// TIA Portal V17 export
// export: Created 2023-05-12T10:40:25.6107869Z, DisplayName Totally Integrated Automation Portal, DisplayVersion V17 Update 4, DisplayName TIA Portal Openness, DisplayVersion V17 Update 4, DisplayName TIA Portal Version Control Interface, DisplayVersion V17, DisplayName STEP 7 Professional, DisplayVersion V17 Update 4, DisplayName STEP 7 Safety, DisplayVersion V17, DisplayName WinCC Advanced / Unified PC, DisplayVersion V17 Update 4
FUNCTION_BLOCK "FB_EM_InputConditioning"   // FB19, LAD
{ S7_Optimized_Access := 'TRUE' }
VERSION : 0.1
// stored: AutoNumber true, CodeModifiedDate 2023-05-12T12:59:41.6492354Z, CompileDate 2023-05-12T12:59:41.6492354Z, CreationDate 2023-05-08T12:19:11.3376827Z, DownloadWithoutReinit false, HandleErrorsWithinBlock false, InterfaceModifiedDate 2023-05-12T12:59:19.7337351Z, IsConsistent true, IsIECCheckEnabled false, IsKnowHowProtected false, IsRetainMemResEnabled false, IsWriteProtected false, LibraryConformanceStatus Warning: The object contains access to global data blocks., MemoryReserve 100, ModifiedDate 2023-05-12T12:59:41.6492354Z, ParameterModified 2022-09-13T10:25:33.4387708Z, PLCSimAdvancedSupport true, SetENOAutomatically false, StructureModified 2023-05-12T12:59:19.7337351Z, UDAEnableTagReadback false
   VAR
      "TT01_TempZasil_K-22/4_Inst" { S7_SetPoint := 'True'} : "FB_CM_MeasurementPoint";
      "TT02_TempPowr_K-22/4_Inst" { S7_SetPoint := 'True'} : "FB_CM_MeasurementPoint";
      TT04_TempPowr_Os_Rzepichy_Inst { S7_SetPoint := 'True'} : "FB_CM_MeasurementPoint";
      TT06_TempPowr_Zabianka_Inst { S7_SetPoint := 'True'} : "FB_CM_MeasurementPoint";
      "PT01_CisnZasil_ K-22/4_Inst" { S7_SetPoint := 'True'} : "FB_CM_MeasurementPoint";
      "PT02_CisnPowr_ K-22/4_Inst" { S7_SetPoint := 'True'} : "FB_CM_MeasurementPoint";
      PT03_CisnZasil_Os_Rzepichy_Inst { S7_SetPoint := 'True'} : "FB_CM_MeasurementPoint";
      PT04_CisnPowr_Os_Rzepichy_Inst { S7_SetPoint := 'True'} : "FB_CM_MeasurementPoint";
      PT05_CisnZasil_Zabianka_Inst { S7_SetPoint := 'True'} : "FB_CM_MeasurementPoint";
      PT06_CisnPowr_Zabianka_Inst { S7_SetPoint := 'True'} : "FB_CM_MeasurementPoint";
      TTs_TempSzafy_Inst { S7_SetPoint := 'True'} : "FB_CM_MeasurementPoint";
      TTk_TempKom_Inst { S7_SetPoint := 'True'} : "FB_CM_MeasurementPoint";
      TTz_TempZewn_Inst { S7_SetPoint := 'True'} : "FB_CM_MeasurementPoint";
      FT01_Przeplyw_Inst { S7_SetPoint := 'True'} : "FB_CM_MeasurementPoint";
      Rezerwa1_Inst { S7_SetPoint := 'True'} : "FB_CM_MeasurementPoint";
      Rezerwa2_Inst { S7_SetPoint := 'True'} : "FB_CM_MeasurementPoint";
   END_VAR
BEGIN

REGION Network 1: TT01_TempZasil_K-22/4 - Temperatura zasilania z K-22/4
   // TT01_TempZasil_K-22/4 - Temperatura zasilania z K-22/4
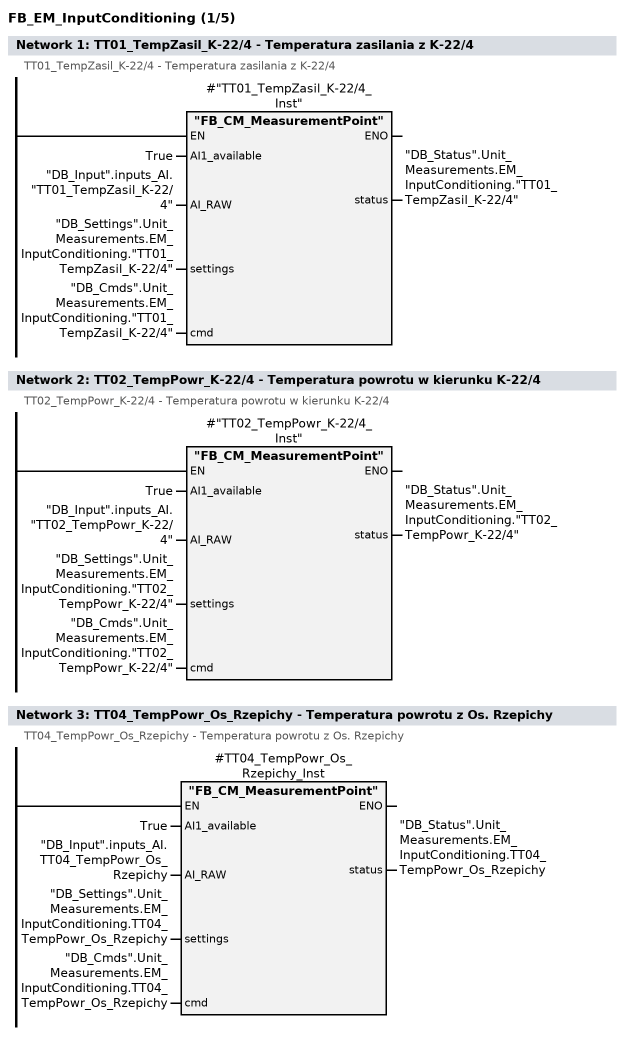
   RUNG wire#powerrail
      #"TT01_TempZasil_K-22/4_Inst"(AI1_available := True, AI_RAW := "DB_Input".inputs_AI."TT01_TempZasil_K-22/4", settings := "DB_Settings".Unit_Measurements.EM_InputConditioning."TT01_TempZasil_K-22/4", cmd := "DB_Cmds".Unit_Measurements.EM_InputConditioning."TT01_TempZasil_K-22/4", status => "DB_Status".Unit_Measurements.EM_InputConditioning."TT01_TempZasil_K-22/4")
   END_RUNG
   // the same network as SCL:
   #"TT01_TempZasil_K-22/4_Inst"(AI1_available := True,   // "FB_CM_MeasurementPoint"
                           AI_RAW := "DB_Input".inputs_AI."TT01_TempZasil_K-22/4",
                           settings := "DB_Settings".Unit_Measurements.EM_InputConditioning."TT01_TempZasil_K-22/4",
                           cmd := "DB_Cmds".Unit_Measurements.EM_InputConditioning."TT01_TempZasil_K-22/4",
                           status => "DB_Status".Unit_Measurements.EM_InputConditioning."TT01_TempZasil_K-22/4");
END_REGION

REGION Network 2: TT02_TempPowr_K-22/4 - Temperatura powrotu w kierunku K-22/4
   // TT02_TempPowr_K-22/4 - Temperatura powrotu w kierunku K-22/4
   RUNG wire#powerrail
      #"TT02_TempPowr_K-22/4_Inst"(AI1_available := True, AI_RAW := "DB_Input".inputs_AI."TT02_TempPowr_K-22/4", settings := "DB_Settings".Unit_Measurements.EM_InputConditioning."TT02_TempPowr_K-22/4", cmd := "DB_Cmds".Unit_Measurements.EM_InputConditioning."TT02_TempPowr_K-22/4", status => "DB_Status".Unit_Measurements.EM_InputConditioning."TT02_TempPowr_K-22/4")
   END_RUNG
   // the same network as SCL:
   #"TT02_TempPowr_K-22/4_Inst"(AI1_available := True,   // "FB_CM_MeasurementPoint"
                           AI_RAW := "DB_Input".inputs_AI."TT02_TempPowr_K-22/4",
                           settings := "DB_Settings".Unit_Measurements.EM_InputConditioning."TT02_TempPowr_K-22/4",
                           cmd := "DB_Cmds".Unit_Measurements.EM_InputConditioning."TT02_TempPowr_K-22/4",
                           status => "DB_Status".Unit_Measurements.EM_InputConditioning."TT02_TempPowr_K-22/4");
END_REGION

REGION Network 3: TT04_TempPowr_Os_Rzepichy - Temperatura powrotu z Os. Rzepichy
   // TT04_TempPowr_Os_Rzepichy - Temperatura powrotu z Os. Rzepichy
   RUNG wire#powerrail
      #TT04_TempPowr_Os_Rzepichy_Inst(AI1_available := True, AI_RAW := "DB_Input".inputs_AI.TT04_TempPowr_Os_Rzepichy, settings := "DB_Settings".Unit_Measurements.EM_InputConditioning.TT04_TempPowr_Os_Rzepichy, cmd := "DB_Cmds".Unit_Measurements.EM_InputConditioning.TT04_TempPowr_Os_Rzepichy, status => "DB_Status".Unit_Measurements.EM_InputConditioning.TT04_TempPowr_Os_Rzepichy)
   END_RUNG
   // the same network as SCL:
   #TT04_TempPowr_Os_Rzepichy_Inst(AI1_available := True,   // "FB_CM_MeasurementPoint"
                           AI_RAW := "DB_Input".inputs_AI.TT04_TempPowr_Os_Rzepichy,
                           settings := "DB_Settings".Unit_Measurements.EM_InputConditioning.TT04_TempPowr_Os_Rzepichy,
                           cmd := "DB_Cmds".Unit_Measurements.EM_InputConditioning.TT04_TempPowr_Os_Rzepichy,
                           status => "DB_Status".Unit_Measurements.EM_InputConditioning.TT04_TempPowr_Os_Rzepichy);
END_REGION

REGION Network 4: TT06_TempPowr_Zabianka - Temperatura powrotu z Żabianka
   // TT06_TempPowr_Zabianka - Temperatura powrotu z Żabianka
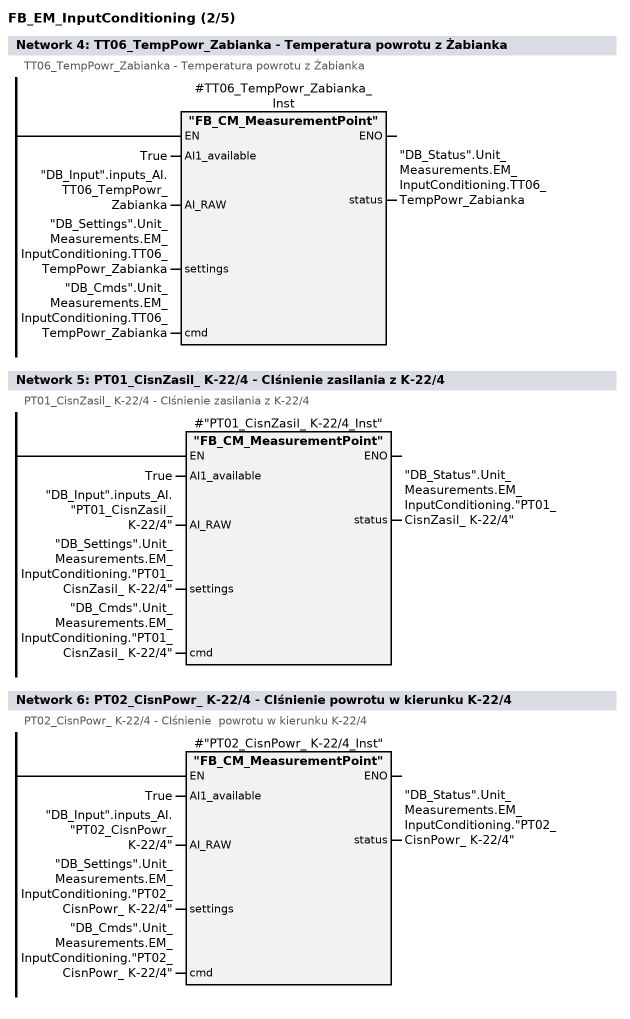
   RUNG wire#powerrail
      #TT06_TempPowr_Zabianka_Inst(AI1_available := True, AI_RAW := "DB_Input".inputs_AI.TT06_TempPowr_Zabianka, settings := "DB_Settings".Unit_Measurements.EM_InputConditioning.TT06_TempPowr_Zabianka, cmd := "DB_Cmds".Unit_Measurements.EM_InputConditioning.TT06_TempPowr_Zabianka, status => "DB_Status".Unit_Measurements.EM_InputConditioning.TT06_TempPowr_Zabianka)
   END_RUNG
   // the same network as SCL:
   #TT06_TempPowr_Zabianka_Inst(AI1_available := True,   // "FB_CM_MeasurementPoint"
                           AI_RAW := "DB_Input".inputs_AI.TT06_TempPowr_Zabianka,
                           settings := "DB_Settings".Unit_Measurements.EM_InputConditioning.TT06_TempPowr_Zabianka,
                           cmd := "DB_Cmds".Unit_Measurements.EM_InputConditioning.TT06_TempPowr_Zabianka,
                           status => "DB_Status".Unit_Measurements.EM_InputConditioning.TT06_TempPowr_Zabianka);
END_REGION

REGION Network 5: PT01_CisnZasil_ K-22/4 - CIśnienie zasilania z K-22/4
   // PT01_CisnZasil_ K-22/4 - CIśnienie zasilania z K-22/4
   RUNG wire#powerrail
      #"PT01_CisnZasil_ K-22/4_Inst"(AI1_available := True, AI_RAW := "DB_Input".inputs_AI."PT01_CisnZasil_ K-22/4", settings := "DB_Settings".Unit_Measurements.EM_InputConditioning."PT01_CisnZasil_ K-22/4", cmd := "DB_Cmds".Unit_Measurements.EM_InputConditioning."PT01_CisnZasil_ K-22/4", status => "DB_Status".Unit_Measurements.EM_InputConditioning."PT01_CisnZasil_ K-22/4")
   END_RUNG
   // the same network as SCL:
   #"PT01_CisnZasil_ K-22/4_Inst"(AI1_available := True,   // "FB_CM_MeasurementPoint"
                           AI_RAW := "DB_Input".inputs_AI."PT01_CisnZasil_ K-22/4",
                           settings := "DB_Settings".Unit_Measurements.EM_InputConditioning."PT01_CisnZasil_ K-22/4",
                           cmd := "DB_Cmds".Unit_Measurements.EM_InputConditioning."PT01_CisnZasil_ K-22/4",
                           status => "DB_Status".Unit_Measurements.EM_InputConditioning."PT01_CisnZasil_ K-22/4");
END_REGION

REGION Network 6: PT02_CisnPowr_ K-22/4 - CIśnienie powrotu w kierunku K-22/4
   // PT02_CisnPowr_ K-22/4 - CIśnienie  powrotu w kierunku K-22/4
   RUNG wire#powerrail
      #"PT02_CisnPowr_ K-22/4_Inst"(AI1_available := True, AI_RAW := "DB_Input".inputs_AI."PT02_CisnPowr_ K-22/4", settings := "DB_Settings".Unit_Measurements.EM_InputConditioning."PT02_CisnPowr_ K-22/4", cmd := "DB_Cmds".Unit_Measurements.EM_InputConditioning."PT02_CisnPowr_ K-22/4", status => "DB_Status".Unit_Measurements.EM_InputConditioning."PT02_CisnPowr_ K-22/4")
   END_RUNG
   // the same network as SCL:
   #"PT02_CisnPowr_ K-22/4_Inst"(AI1_available := True,   // "FB_CM_MeasurementPoint"
                           AI_RAW := "DB_Input".inputs_AI."PT02_CisnPowr_ K-22/4",
                           settings := "DB_Settings".Unit_Measurements.EM_InputConditioning."PT02_CisnPowr_ K-22/4",
                           cmd := "DB_Cmds".Unit_Measurements.EM_InputConditioning."PT02_CisnPowr_ K-22/4",
                           status => "DB_Status".Unit_Measurements.EM_InputConditioning."PT02_CisnPowr_ K-22/4");
END_REGION

REGION Network 7: PT03_CisnZasil_Os_Rzepichy - Ciśnienie zasilania w kierunku Os. Rzepichy
   // PT03_CisnZasil_Os_Rzepichy - Ciśnienie zasilania w kierunku Os. Rzepichy
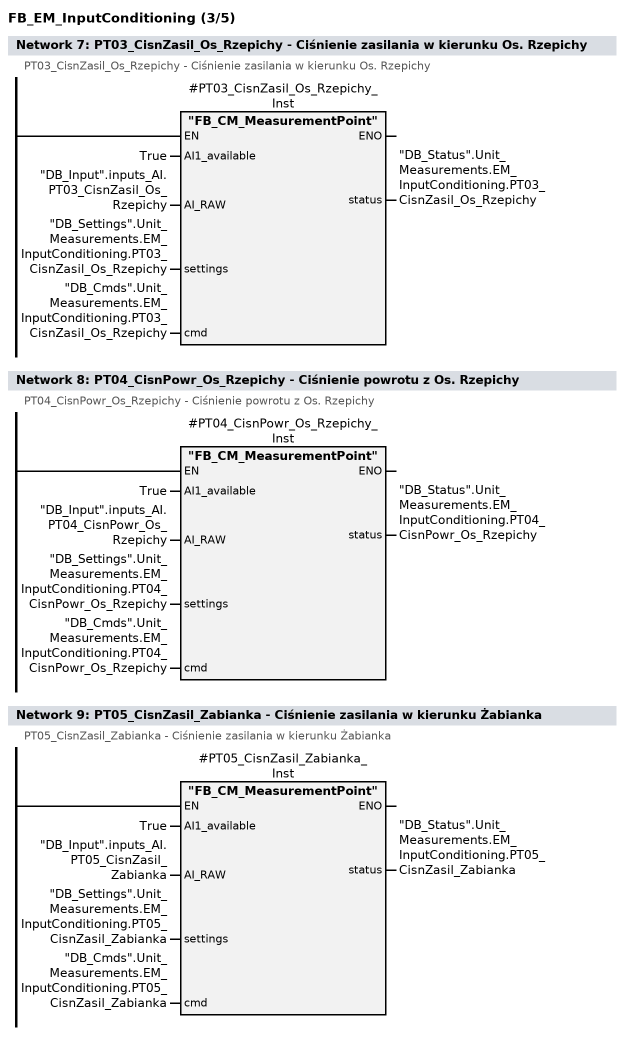
   RUNG wire#powerrail
      #PT03_CisnZasil_Os_Rzepichy_Inst(AI1_available := True, AI_RAW := "DB_Input".inputs_AI.PT03_CisnZasil_Os_Rzepichy, settings := "DB_Settings".Unit_Measurements.EM_InputConditioning.PT03_CisnZasil_Os_Rzepichy, cmd := "DB_Cmds".Unit_Measurements.EM_InputConditioning.PT03_CisnZasil_Os_Rzepichy, status => "DB_Status".Unit_Measurements.EM_InputConditioning.PT03_CisnZasil_Os_Rzepichy)
   END_RUNG
   // the same network as SCL:
   #PT03_CisnZasil_Os_Rzepichy_Inst(AI1_available := True,   // "FB_CM_MeasurementPoint"
                           AI_RAW := "DB_Input".inputs_AI.PT03_CisnZasil_Os_Rzepichy,
                           settings := "DB_Settings".Unit_Measurements.EM_InputConditioning.PT03_CisnZasil_Os_Rzepichy,
                           cmd := "DB_Cmds".Unit_Measurements.EM_InputConditioning.PT03_CisnZasil_Os_Rzepichy,
                           status => "DB_Status".Unit_Measurements.EM_InputConditioning.PT03_CisnZasil_Os_Rzepichy);
END_REGION

REGION Network 8: PT04_CisnPowr_Os_Rzepichy - Ciśnienie powrotu z Os. Rzepichy
   // PT04_CisnPowr_Os_Rzepichy - Ciśnienie powrotu z Os. Rzepichy
   RUNG wire#powerrail
      #PT04_CisnPowr_Os_Rzepichy_Inst(AI1_available := True, AI_RAW := "DB_Input".inputs_AI.PT04_CisnPowr_Os_Rzepichy, settings := "DB_Settings".Unit_Measurements.EM_InputConditioning.PT04_CisnPowr_Os_Rzepichy, cmd := "DB_Cmds".Unit_Measurements.EM_InputConditioning.PT04_CisnPowr_Os_Rzepichy, status => "DB_Status".Unit_Measurements.EM_InputConditioning.PT04_CisnPowr_Os_Rzepichy)
   END_RUNG
   // the same network as SCL:
   #PT04_CisnPowr_Os_Rzepichy_Inst(AI1_available := True,   // "FB_CM_MeasurementPoint"
                           AI_RAW := "DB_Input".inputs_AI.PT04_CisnPowr_Os_Rzepichy,
                           settings := "DB_Settings".Unit_Measurements.EM_InputConditioning.PT04_CisnPowr_Os_Rzepichy,
                           cmd := "DB_Cmds".Unit_Measurements.EM_InputConditioning.PT04_CisnPowr_Os_Rzepichy,
                           status => "DB_Status".Unit_Measurements.EM_InputConditioning.PT04_CisnPowr_Os_Rzepichy);
END_REGION

REGION Network 9: PT05_CisnZasil_Zabianka - Ciśnienie zasilania w kierunku Żabianka
   // PT05_CisnZasil_Zabianka - Ciśnienie zasilania w kierunku Żabianka
   RUNG wire#powerrail
      #PT05_CisnZasil_Zabianka_Inst(AI1_available := True, AI_RAW := "DB_Input".inputs_AI.PT05_CisnZasil_Zabianka, settings := "DB_Settings".Unit_Measurements.EM_InputConditioning.PT05_CisnZasil_Zabianka, cmd := "DB_Cmds".Unit_Measurements.EM_InputConditioning.PT05_CisnZasil_Zabianka, status => "DB_Status".Unit_Measurements.EM_InputConditioning.PT05_CisnZasil_Zabianka)
   END_RUNG
   // the same network as SCL:
   #PT05_CisnZasil_Zabianka_Inst(AI1_available := True,   // "FB_CM_MeasurementPoint"
                           AI_RAW := "DB_Input".inputs_AI.PT05_CisnZasil_Zabianka,
                           settings := "DB_Settings".Unit_Measurements.EM_InputConditioning.PT05_CisnZasil_Zabianka,
                           cmd := "DB_Cmds".Unit_Measurements.EM_InputConditioning.PT05_CisnZasil_Zabianka,
                           status => "DB_Status".Unit_Measurements.EM_InputConditioning.PT05_CisnZasil_Zabianka);
END_REGION

REGION Network 10: PT06_CisnPowr_Zabianka - Ciśnienie powrotu z Żabianka
   // PT06_CisnPowr_Zabianka - Ciśnienie powrotu z Żabianka
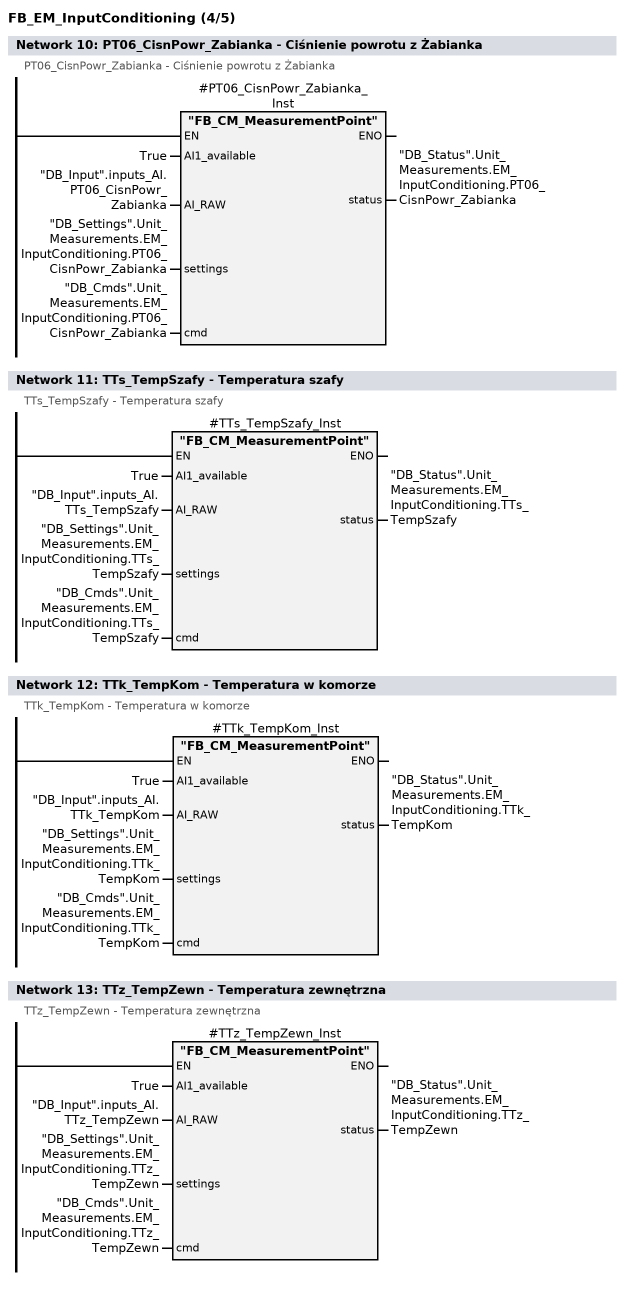
   RUNG wire#powerrail
      #PT06_CisnPowr_Zabianka_Inst(AI1_available := True, AI_RAW := "DB_Input".inputs_AI.PT06_CisnPowr_Zabianka, settings := "DB_Settings".Unit_Measurements.EM_InputConditioning.PT06_CisnPowr_Zabianka, cmd := "DB_Cmds".Unit_Measurements.EM_InputConditioning.PT06_CisnPowr_Zabianka, status => "DB_Status".Unit_Measurements.EM_InputConditioning.PT06_CisnPowr_Zabianka)
   END_RUNG
   // the same network as SCL:
   #PT06_CisnPowr_Zabianka_Inst(AI1_available := True,   // "FB_CM_MeasurementPoint"
                           AI_RAW := "DB_Input".inputs_AI.PT06_CisnPowr_Zabianka,
                           settings := "DB_Settings".Unit_Measurements.EM_InputConditioning.PT06_CisnPowr_Zabianka,
                           cmd := "DB_Cmds".Unit_Measurements.EM_InputConditioning.PT06_CisnPowr_Zabianka,
                           status => "DB_Status".Unit_Measurements.EM_InputConditioning.PT06_CisnPowr_Zabianka);
END_REGION

REGION Network 11: TTs_TempSzafy - Temperatura szafy
   // TTs_TempSzafy - Temperatura szafy
   RUNG wire#powerrail
      #TTs_TempSzafy_Inst(AI1_available := True, AI_RAW := "DB_Input".inputs_AI.TTs_TempSzafy, settings := "DB_Settings".Unit_Measurements.EM_InputConditioning.TTs_TempSzafy, cmd := "DB_Cmds".Unit_Measurements.EM_InputConditioning.TTs_TempSzafy, status => "DB_Status".Unit_Measurements.EM_InputConditioning.TTs_TempSzafy)
   END_RUNG
   // the same network as SCL:
   #TTs_TempSzafy_Inst(AI1_available := True,   // "FB_CM_MeasurementPoint"
                       AI_RAW := "DB_Input".inputs_AI.TTs_TempSzafy,
                       settings := "DB_Settings".Unit_Measurements.EM_InputConditioning.TTs_TempSzafy,
                       cmd := "DB_Cmds".Unit_Measurements.EM_InputConditioning.TTs_TempSzafy,
                       status => "DB_Status".Unit_Measurements.EM_InputConditioning.TTs_TempSzafy);
END_REGION

REGION Network 12: TTk_TempKom - Temperatura w komorze
   // TTk_TempKom - Temperatura w komorze
   RUNG wire#powerrail
      #TTk_TempKom_Inst(AI1_available := True, AI_RAW := "DB_Input".inputs_AI.TTk_TempKom, settings := "DB_Settings".Unit_Measurements.EM_InputConditioning.TTk_TempKom, cmd := "DB_Cmds".Unit_Measurements.EM_InputConditioning.TTk_TempKom, status => "DB_Status".Unit_Measurements.EM_InputConditioning.TTk_TempKom)
   END_RUNG
   // the same network as SCL:
   #TTk_TempKom_Inst(AI1_available := True,   // "FB_CM_MeasurementPoint"
                     AI_RAW := "DB_Input".inputs_AI.TTk_TempKom,
                     settings := "DB_Settings".Unit_Measurements.EM_InputConditioning.TTk_TempKom,
                     cmd := "DB_Cmds".Unit_Measurements.EM_InputConditioning.TTk_TempKom,
                     status => "DB_Status".Unit_Measurements.EM_InputConditioning.TTk_TempKom);
END_REGION

REGION Network 13: TTz_TempZewn - Temperatura zewnętrzna
   // TTz_TempZewn - Temperatura zewnętrzna
   RUNG wire#powerrail
      #TTz_TempZewn_Inst(AI1_available := True, AI_RAW := "DB_Input".inputs_AI.TTz_TempZewn, settings := "DB_Settings".Unit_Measurements.EM_InputConditioning.TTz_TempZewn, cmd := "DB_Cmds".Unit_Measurements.EM_InputConditioning.TTz_TempZewn, status => "DB_Status".Unit_Measurements.EM_InputConditioning.TTz_TempZewn)
   END_RUNG
   // the same network as SCL:
   #TTz_TempZewn_Inst(AI1_available := True,   // "FB_CM_MeasurementPoint"
                      AI_RAW := "DB_Input".inputs_AI.TTz_TempZewn,
                      settings := "DB_Settings".Unit_Measurements.EM_InputConditioning.TTz_TempZewn,
                      cmd := "DB_Cmds".Unit_Measurements.EM_InputConditioning.TTz_TempZewn,
                      status => "DB_Status".Unit_Measurements.EM_InputConditioning.TTz_TempZewn);
END_REGION

REGION Network 14: FT01_Przeplyw - Przepływ
   // FT01_Przeplyw - Przepływ
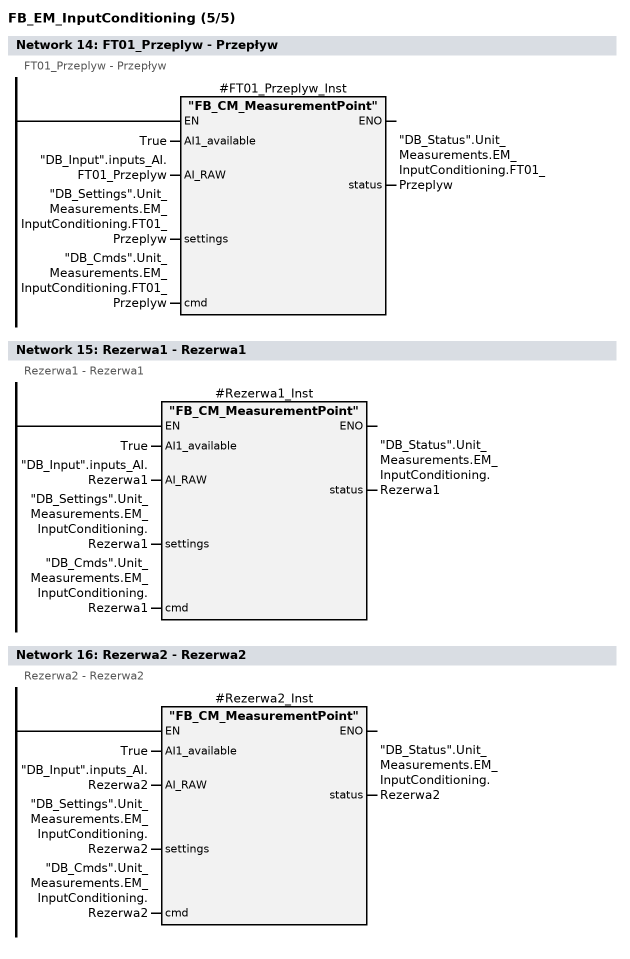
   RUNG wire#powerrail
      #FT01_Przeplyw_Inst(AI1_available := True, AI_RAW := "DB_Input".inputs_AI.FT01_Przeplyw, settings := "DB_Settings".Unit_Measurements.EM_InputConditioning.FT01_Przeplyw, cmd := "DB_Cmds".Unit_Measurements.EM_InputConditioning.FT01_Przeplyw, status => "DB_Status".Unit_Measurements.EM_InputConditioning.FT01_Przeplyw)
   END_RUNG
   // the same network as SCL:
   #FT01_Przeplyw_Inst(AI1_available := True,   // "FB_CM_MeasurementPoint"
                       AI_RAW := "DB_Input".inputs_AI.FT01_Przeplyw,
                       settings := "DB_Settings".Unit_Measurements.EM_InputConditioning.FT01_Przeplyw,
                       cmd := "DB_Cmds".Unit_Measurements.EM_InputConditioning.FT01_Przeplyw,
                       status => "DB_Status".Unit_Measurements.EM_InputConditioning.FT01_Przeplyw);
END_REGION

REGION Network 15: Rezerwa1 - Rezerwa1
   // Rezerwa1 - Rezerwa1
   RUNG wire#powerrail
      #Rezerwa1_Inst(AI1_available := True, AI_RAW := "DB_Input".inputs_AI.Rezerwa1, settings := "DB_Settings".Unit_Measurements.EM_InputConditioning.Rezerwa1, cmd := "DB_Cmds".Unit_Measurements.EM_InputConditioning.Rezerwa1, status => "DB_Status".Unit_Measurements.EM_InputConditioning.Rezerwa1)
   END_RUNG
   // the same network as SCL:
   #Rezerwa1_Inst(AI1_available := True,   // "FB_CM_MeasurementPoint"
                  AI_RAW := "DB_Input".inputs_AI.Rezerwa1,
                  settings := "DB_Settings".Unit_Measurements.EM_InputConditioning.Rezerwa1,
                  cmd := "DB_Cmds".Unit_Measurements.EM_InputConditioning.Rezerwa1,
                  status => "DB_Status".Unit_Measurements.EM_InputConditioning.Rezerwa1);
END_REGION

REGION Network 16: Rezerwa2 - Rezerwa2
   // Rezerwa2 - Rezerwa2
   RUNG wire#powerrail
      #Rezerwa2_Inst(AI1_available := True, AI_RAW := "DB_Input".inputs_AI.Rezerwa2, settings := "DB_Settings".Unit_Measurements.EM_InputConditioning.Rezerwa2, cmd := "DB_Cmds".Unit_Measurements.EM_InputConditioning.Rezerwa2, status => "DB_Status".Unit_Measurements.EM_InputConditioning.Rezerwa2)
   END_RUNG
   // the same network as SCL:
   #Rezerwa2_Inst(AI1_available := True,   // "FB_CM_MeasurementPoint"
                  AI_RAW := "DB_Input".inputs_AI.Rezerwa2,
                  settings := "DB_Settings".Unit_Measurements.EM_InputConditioning.Rezerwa2,
                  cmd := "DB_Cmds".Unit_Measurements.EM_InputConditioning.Rezerwa2,
                  status => "DB_Status".Unit_Measurements.EM_InputConditioning.Rezerwa2);
END_REGION
END_FUNCTION_BLOCK
